# EPICS StreamDevice protocol: drvMegampApp/Db/Megamp.proto
OutTerminator = CR LF;
InTerminator = LF CR;

rd_attr {
   out "*\$1C\$2A\$3";
   in "OK %i";
}

wr_attr {
   out "*\$1C\$2A\$3,%i";
   in "OK";
   @init { rd_attr; }
}

#sel_channel {
#   out "*%(A)iC%(B)iA0";
#   in "OK %*i"
#}

# Connect a stringout record to this to get
# a generic command interface.
# After processing finishes, the record contains the reply.

debug {
    ExtraInput = Ignore;
    out "%s"; in "%39c"
}
